Yaskawa INFORM job: MOVC_DEMO.JBI

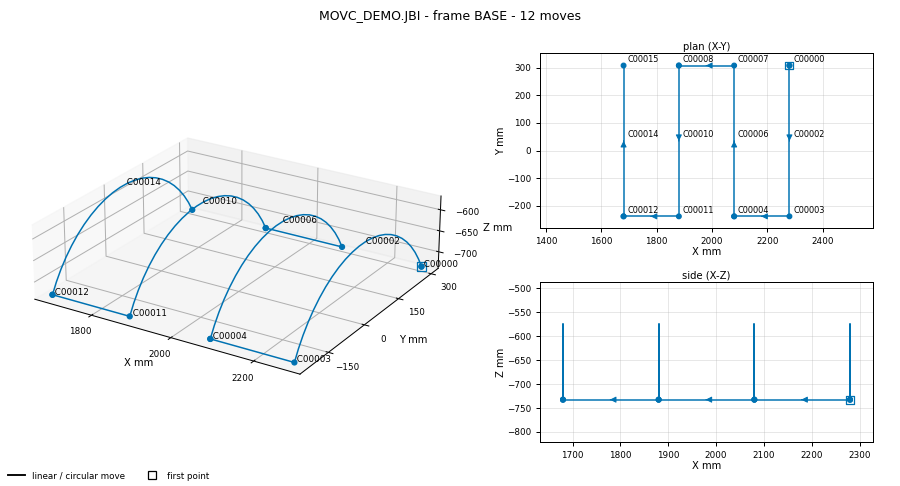
[picture p0: tool path of MOVC_DEMO.JBI in frame BASE, 12 of 16 moves have a stored position in this frame; points joined in program order, loops and branches not executed]
/JOB
//NAME MOVC_DEMO
//POS
///NPOS 16,0,0,0,0,0
///TOOL 0
///POSTYPE BASE
///RECTAN
///RCONF 0,0,0,0,0,0,0,0,0,0,0,0,0,0,0,0,0,0,0,0,0,0,0,0
C00000=2280.000,307.798,-732.500,120.0000,0.0000,0.0000
C00001=2280.000,307.798,-732.500,120.0000,0.0000,0.0000
C00002=2280.000,35.000,-575.000,180.0000,0.0000,0.0000
C00003=2280.000,-237.798,-732.500,240.0000,0.0000,0.0000
C00004=2080.000,-237.798,-732.500,240.0000,0.0000,0.0000
C00005=2080.000,-237.798,-732.500,240.0000,0.0000,0.0000
C00006=2080.000,35.000,-575.000,180.0000,0.0000,0.0000
C00007=2080.000,307.798,-732.500,120.0000,0.0000,0.0000
C00008=1880.000,307.798,-732.500,120.0000,0.0000,0.0000
C00009=1880.000,307.798,-732.500,120.0000,0.0000,0.0000
C00010=1880.000,35.000,-575.000,180.0000,0.0000,0.0000
C00011=1880.000,-237.798,-732.500,240.0000,0.0000,0.0000
C00012=1680.000,-237.798,-732.500,240.0000,0.0000,0.0000
C00013=1680.000,-237.798,-732.500,240.0000,0.0000,0.0000
C00014=1680.000,35.000,-575.000,180.0000,0.0000,0.0000
C00015=1680.000,307.798,-732.500,120.0000,0.0000,0.0000
//INST
///DATE 2023/03/27 17:16
///ATTR SC,RW,RJ
////FRAME BASE
///GROUP1 RB1
NOP
MOVJ C00000 VJ=12.00
MOVC C00001 V=100.0
MOVC C00002 V=100.0
MOVC C00003 V=100.0
MOVL C00004 V=100.0
MOVC C00005 V=100.0
MOVC C00006 V=100.0
MOVC C00007 V=100.0
MOVL C00008 V=100.0
MOVC C00009 V=100.0
MOVC C00010 V=100.0
MOVC C00011 V=100.0
MOVL C00012 V=100.0
MOVC C00013 V=100.0
MOVC C00014 V=100.0
MOVC C00015 V=100.0
END
